// Mitsubishi GX Works2 project: m01   PLC: Q02/Q02H

PROGRAM MAIN
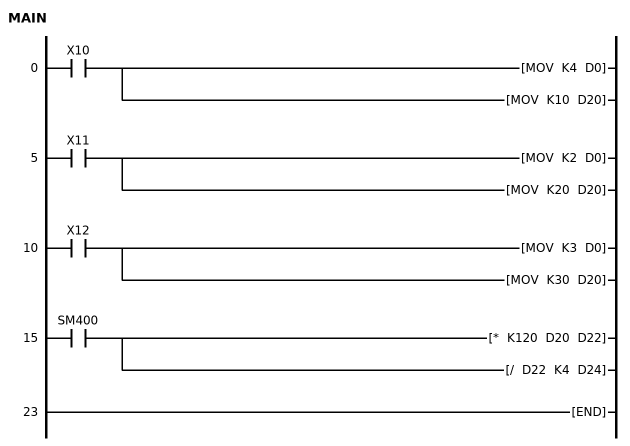
0     LD      X10
      MOV     K4 D0
      MOV     K10 D20
5     LD      X11
      MOV     K2 D0
      MOV     K20 D20
10    LD      X12
      MOV     K3 D0
      MOV     K30 D20
15    LD      SM400
      *       K120 D20 D22
      /       D22 K4 D24
23    END
END_PROGRAM
